// Author: Feijian Ni
// Date: 2024.11.26
FUNCTION_BLOCK FB_RedunJntControl_202504

VAR
	// joint 6 deviation from center
	m_jnt6Bias :LREAL;
	
	// static velocity threshold
	m_staticWVelThres :LREAL := 10 *g_deg2Rad;
	m_staticVelThres :LREAL := 0.02;
	m_staticTime:LREAL:=0;
	m_staticTimeThres:LREAL:=0.5;

	// rudundancy track flag
	m_trackFlag :BOOL;
	
	// orientation nullspace jacobian
	m_oriNullJaco: Mat4d;
	
	// current manipulation velocity
	m_curManipWVel :LREAL :=0;
	m_curManipVel:LREAL:=0;
	
	// joint4 dynamic limit and limit buffer
	m_jntPosUb, m_jntPosLb:LREAL;
	m_jntUpLimit,m_jntLowLimit:LREAL;
	m_targetVelUb, m_targetVelLb:LREAL;
	m_jntLimitBuffer : LREAL :=2*g_deg2Rad;
	
	// scale near singularity
	m_singScale:LREAL;
	
	// control paramters for redundant joint4 position control
//	m_redunJntKp: LREAL:=8.0;
//	m_redunJntKd:LREAL:=0.2;
//	m_redunJntKp: LREAL:=3.0;
//	m_redunJntKd:LREAL:=0.1;
	m_redunJntKp: LREAL:=40;
	m_redunJntKd:LREAL:=2;
	m_redunJntKi:LREAL:=0;
	m_redunJntKiLimit: LREAL:=200;
	m_redunJntCtrlLimit:LREAL:=500;

	// redundant track parameters
	m_redunKp:LREAL:=6;
	m_deadband :LREAL := 2*g_deg2rad;
	m_minDeadband:LREAL:=2*g_deg2rad;
	m_maxDeadband:LREAL:=20*g_deg2rad;
	m_maxCmdPosErr:LREAL:=5*g_deg2rad;
	m_maxCmdVel :LREAL := 15;
	m_maxJntAcc :LREAL := 30;
	m_targetJntVel:LREAL;
	
	// command joint4 position and veloicty in motor for next cycle
	m_cmdJntPos: LREAL;
	m_cmdJntVel: LREAL;
	m_cmdJntAcc: LREAL;

	// PID for joint position
	m_jntPIDCtrl: FB_PID;
	m_jntCtrlTrq: LREAL;
	
	// static duration
	m_curStaticDuration :LREAL:=0;
	m_staticDurationThres :LREAL :=0.1;

END_VAR

METHOD calcDynaLimit : BOOL
VAR_IN_OUT CONSTANT
	i_masterArm :FB_MasterArm;
END_VAR
VAR
		curLinkPos:LREAL;
		scale:LREAL;
END_VAR
// structure position limit check
m_jntPosUb:=i_masterArm.jnt4LinkToMotor(i_masterArm.curJntPos[2],i_masterArm.curJntPos[3],
						 m_jntUpLimit-m_jntLimitBuffer);
m_jntPosLb:=i_masterArm.jnt4LinkToMotor(i_masterArm.curJntPos[2],i_masterArm.curJntPos[3],
						 m_jntLowLimit+m_jntLimitBuffer);
						 
// position limit in case joint4 is blocked
m_jntPosUb := MIN(m_jntPosUb, i_masterArm.curJntPos[4]+MIN(m_maxCmdPosErr,ABS(m_jnt6Bias))); 
m_jntPosLb := MAX(m_jntPosLb, i_masterArm.curJntPos[4]-MIN(m_maxCmdPosErr,ABS(m_jnt6Bias))); 

// in case current joint position is out of limit
m_jntPosUb := MAX(m_jntPosUb, i_masterArm.curJntPos[4]); 
m_jntPosLb := MIN(m_jntPosLb, i_masterArm.curJntPos[4]); 

// velocity limit 
m_targetVelUb:= MIN(m_maxCmdVel, SQRT(2*m_maxJntAcc* ABS(m_jntPosUb-m_cmdJntPos)));
m_targetVelLb:= MAX(-m_maxCmdVel, -SQRT(2*m_maxJntAcc* ABS(m_jntPosLb-m_cmdJntPos)));
END_METHOD

METHOD PROTECTED calcJnt6Bias : LREAL
VAR_IN_OUT CONSTANT
	i_masterArm :FB_MasterArm;
END_VAR
IF 1= i_masterArm.armIdx THEN
	calcJnt6Bias :=i_masterArm.curJntPos[6]+PI/2;
ELSE 
	calcJnt6Bias := i_masterArm.curJntPos[6]-PI/2;
END_IF
END_METHOD

// calculate orientation manipulation velocity(in local coordinate)
METHOD calcManipVel : BOOL
VAR_IN_OUT CONSTANT
	i_masterArm :FB_MasterArm;
END_VAR
VAR
	vel:Vec3d;
	wVelWrd,wVelLocal:Vec3d;
	rotT:Mat3d;
END_VAR
vel[1]:= i_masterArm.m_curCartLinkTwist[1];
vel[2]:= i_masterArm.m_curCartLinkTwist[2];
vel[3]:= i_masterArm.m_curCartLinkTwist[3];
m_curManipVel:=norm(vel);

wVelWrd[1]:= i_masterArm.m_curCartLinkTwist[4];
wVelWrd[2]:= i_masterArm.m_curCartLinkTwist[5];
wVelWrd[3]:= i_masterArm.m_curCartLinkTwist[6];

matTranspose(i_masterArm.m_curCartLinkPose.m_rot, rotT);
matMultiVec(rotT, wVelWrd, wVelLocal);

wVelLocal[3]:=0;
m_curManipWVel:=norm(wVelLocal);
END_METHOD

METHOD PROTECTED calcNullJaco : Mat4d;
VAR_IN_OUT CONSTANT
	i_masterArm :FB_MasterArm;
END_VAR
VAR
	i,j:INT;
	oriJaco:Mat34;
	oriJt:Mat43;
	oriJJt:Mat3d;
	oriJJtInv:Mat3d;
	oriJPinv:Mat43;
	JpinvJ :Mat4d;
	eye4d :Mat4d := g_eye4d;
END_VAR
// compute pinv of orientation jacobian
FOR i:=1 TO 3 DO
	FOR j:=1 TO 4 DO
		oriJaco[i,j]:=i_masterArm.simJaco[i+3,j+3];
	END_FOR
END_FOR
matTranspose(oriJaco, oriJt);
matMultiply(oriJaco ,oriJt , oriJJt);
invMat3(oriJJt, oriJJtInv);
matMultiply(oriJt, oriJJtInv, oriJPinv);

// calculate nullspace
matMultiply(oriJPinv, oriJaco, JpinvJ);
matSub(eye4d , JpinvJ, calcNullJaco);
END_METHOD

METHOD cmdReduntJntVel : LREAL
VAR_IN_OUT CONSTANT
	i_masterArm :FB_MasterArm;
END_VAR
VAR
	biasVel:LREAL;
	ffVel:LREAL;

END_VAR
// velocity from joint6 bias
IF ABS(m_oriNullJaco[1,1])<g_smallNum THEN
	m_singScale :=0;
ELSE
	m_singScale := MIN(1.0, ABS(m_oriNullJaco[3,1]/m_oriNullJaco[1,1]));
END_IF

m_deadband:=abs(COS(i_masterArm.curJntPos[5]-pi));
m_deadband := m_maxDeadband-(m_maxDeadband-m_minDeadband)*m_deadband;

IF ABS(m_jnt6Bias)>m_deadband THEN
	cmdReduntJntVel:=-1*(m_jnt6Bias-sign(m_jnt6Bias)*m_deadband)*m_redunKp*ABS(m_singScale);
ELSE
	cmdReduntJntVel :=0;
END_IF
END_METHOD

METHOD init : BOOL
VAR_IN_OUT CONSTANT
	i_masterArm :FB_MasterArm;
END_VAR
VAR
	currentRatioMotor2Jnt:LREAL;
END_VAR
m_cmdJntPos:=i_masterArm.curJntPos[4];
m_cmdJntVel:=0;
m_curStaticDuration:=0;

// init controller
currentRatioMotor2Jnt:=GVL_ArmJointParameters.g_motorTrqConst[4]*GVL_ArmJointParameters.g_motorReduction[4]/1000;
m_jntPIDCtrl.init(g_armCtrlCycleTime,m_redunJntKp,m_redunJntKd,m_redunJntKi,
		m_redunJntKiLimit* currentRatioMotor2Jnt,	m_redunJntCtrlLimit*currentRatioMotor2Jnt);

// determin joint limit
IF i_masterArm.armIdx=1 THEN
	m_jntUpLimit := -pi + 15*g_deg2rad;
	m_jntLowLimit := GVL_ArmJointParameters.g_minJntPos[i_masterArm.armIdx,4];
ELSE
	m_jntUpLimit := GVL_ArmJointParameters.g_maxJntPos[i_masterArm.armIdx,4];
	m_jntLowLimit :=0 - 15 *g_deg2rad;
END_IF
END_METHOD

METHOD run : LREAL
VAR_IN_OUT CONSTANT
	i_masterArm :FB_MasterArm;
END_VAR
VAR_INPUT
	i_followEnable :BOOL;
END_VAR


VAR
	velScale,limitScale:LREAL;
	maxAcc, minDec:LREAL;
	wVel:Vec3d;
END_VAR
// joint 6 deviation from center
m_jnt6Bias := calcJnt6Bias(i_masterArm);

// calculate nullspace jacobian
m_oriNullJaco := calcNullJaco(i_masterArm);

// calculate manipulation angular velocity(exclude roll velocity)
 calcManipVel(i_masterArm);

// check if arm is static
m_trackFlag:=startTrackCheck(i_masterArm);

// redundant tracking velocity
IF m_trackFlag THEN
	m_targetJntVel := cmdReduntJntVel(i_masterArm);
	maxAcc := m_maxJntAcc;
ELSE
	m_targetJntVel :=0;
	maxAcc := m_maxJntAcc/3.0;
END_IF

// dynamic limit 
calcDynaLimit(i_masterArm);
m_targetJntVel := LIMIT(m_targetVelLb, m_targetJntVel, m_targetVelUb);

// integrate to get position
m_cmdJntAcc := LIMIT(-maxAcc, (m_targetJntVel - m_cmdJntVel)*g_armCtrlFreq, maxAcc);
m_cmdJntPos:= m_cmdJntPos + m_cmdJntVel * g_armCtrlCycleTime + 0.5*m_cmdJntAcc*g_armCtrlCycleTime*g_armCtrlCycleTime;
m_cmdJntVel := m_cmdJntVel + m_cmdJntAcc *g_armCtrlCycleTime;
m_cmdJntVel:=LIMIT(m_targetVelLb, m_cmdJntVel, m_targetVelUb);

IF m_cmdJntPos >m_jntPosUb AND m_cmdJntVel>0  THEN
	m_cmdJntPos:=m_jntPosUb;
	m_cmdJntVel:=0;
	m_cmdJntAcc:=0;
ELSIF m_cmdJntPos <m_jntPosLb AND m_cmdJntVel<0 THEN
	m_cmdJntPos:=m_jntPosLb;
	m_cmdJntVel:=0;
	m_cmdJntAcc:=0;
END_IF
m_cmdJntPos:=LIMIT(m_jntPosLb, m_cmdJntPos, m_jntPosUb);

// joint position control torque control
m_jntCtrlTrq:=m_jntPIDCtrl.run(m_cmdJntPos,i_masterArm.curJntPos[4], m_cmdJntVel, i_masterArm.curJntVel[4]);
run:=m_jntCtrlTrq;
END_METHOD

METHOD startTrackCheck : BOOL
VAR_IN_OUT CONSTANT
	i_masterArm :FB_MasterArm;
END_VAR
VAR
	jntVelCheck:Vec3d;
END_VAR
IF NOT m_trackFlag THEN
	m_curStaticDuration := m_curStaticDuration + g_armCtrlCycleTime;
	IF m_curStaticDuration < m_staticDurationThres THEN
		startTrackCheck:=FALSE;
		RETURN;
	END_IF
ELSE
	m_curStaticDuration := 0;
END_IF

jntVelCheck[1] := i_masterArm.curJntVel[5];
jntVelCheck[2] := i_masterArm.curJntVel[6];
jntVelCheck[3] := i_masterArm.curJntVel[7];

IF (m_curManipWVel<m_staticWVelThres OR norm(jntVelCheck)< m_staticWVelThres) and m_curManipVel<m_staticVelThres THEN
	m_staticTime:=m_staticTime+g_armCtrlCycleTime;
ELSE
	m_staticTime:=0;
END_IF
startTrackCheck:=m_staticTime<m_staticTimeThres;
END_METHOD

END_FUNCTION_BLOCK

(* stored: Version 1.1.0.1, ProductVersion 3.1.4024.11
   POU FB_RedunJntControl_202504: Id {2da14c1b-ef6b-4c54-8597-76647219be88}, SpecialFunc None
   Method calcDynaLimit: Id {90e0b621-165c-4a1a-93c3-1fdb42db1d7e}
   Method calcJnt6Bias: Id {4f19ec43-caf1-43d1-8297-5cc8aee7dd76}
   Method calcManipVel: Id {ab8f8c50-76d8-4070-aeb0-40f16d9ade59}
   Method calcNullJaco: Id {7b66e0fa-0d62-4f5d-b303-077cc17d9b4d}
   Method cmdReduntJntVel: Id {1a06e4a7-636c-4122-967e-2c3678acbb33}
   Method init: Id {bedc279c-107c-48ba-8160-b8ed00ba098f}
   Method run: Id {69800672-31dd-4dd3-afe5-ecd9f2cc2c4c}
   Method startTrackCheck: Id {5a32f58f-1006-41c3-85cb-4b82e3a95bfa} *)
